ABB RAPID module: Target_R.mod

MODULE Target_R
    CONST robtarget TG_pick:=[[177.042141649,-272.000801516,190.000004036],[0.000000058,0.923879576,0.000000285,0.382683327],[0,-2,-1,4],[-107.239308648,9E+09,9E+09,9E+09,9E+09,9E+09]];
    CONST robtarget pick_up:=[[100.000104042,-278.500207981,150.000028222],[-0.000000126,-0.707106773,0.707106789,0.000000032],[0,-2,-1,4],[-101.964426672,9E+09,9E+09,9E+09,9E+09,9E+09]];
    CONST robtarget pick:=[[100,-278.5,50.43],[0,-0.707106781,0.707106781,0],[0,-2,-1,4],[-101.964426261,9E+09,9E+09,9E+09,9E+09,9E+09]];
    CONST robtarget check_BFR:=[[337.65,-25.09,414.16],[0.47949,-0.522281,0.486899,0.510138],[1,0,-1,4],[-166.865,9E+09,9E+09,9E+09,9E+09,9E+09]];
    CONST robtarget check_R:=[[352.06,-3.78,414.93],[0.468537,-0.49966,-0.504407,0.525725],[1,0,-2,4],[171.664,9E+09,9E+09,9E+09,9E+09,9E+09]];
    CONST robtarget TG_waitpoint:=[[260.000500472,-88.346067188,381.139966328],[0.499999312,-0.500000007,0.500000478,0.500000203],[0,0,-2,4],[-157.417353478,9E+09,9E+09,9E+09,9E+09,9E+09]];
    CONST robtarget waitpoint:=[[320.000617334,-110.201098524,199.999425349],[0.499999098,-0.500000027,0.500000616,0.50000026],[1,0,-1,4],[-162.867770325,9E+09,9E+09,9E+09,9E+09,9E+09]];
    CONST robtarget center:=[[320.000394297,-24.06071977,199.999617271],[0.499999361,-0.499999966,0.500000448,0.500000224],[1,0,-2,4],[-162.867771789,9E+09,9E+09,9E+09,9E+09,9E+09]];
    CONST robtarget home:=[[89.387954365,-156.622115869,147.913470331],[0.066010721,-0.842420916,-0.111214905,-0.523068666],[0,0,0,4],[-101.964426493,9E+09,9E+09,9E+09,9E+09,9E+09]];
    CONST robtarget TG_case_1:=[[320,-35.2,200],[0.5,-0.5,0.5,0.5],[1,0,-1,4],[-162.867772063,9E+09,9E+09,9E+09,9E+09,9E+09]];
    CONST robtarget TG_case_1_2:=[[285,-0.2,200],[0.707106781,0,0.707106781,0],[1,1,1,4],[-162.867775031,9E+09,9E+09,9E+09,9E+09,9E+09]];
    CONST robtarget TG_case_1_3:=[[250.000130819,-0.200197514,199.999945575],[0.707106719,-0.000000126,0.707106844,-0.000000064],[1,1,1,4],[-162.867770883,9E+09,9E+09,9E+09,9E+09,9E+09]];
    CONST robtarget TG_case_1_4:=[[250.000195865,-100.200387425,199.999831039],[0.707106608,-0.000000212,0.707106955,-0.000000105],[1,1,1,4],[-162.867770415,9E+09,9E+09,9E+09,9E+09,9E+09]];
    CONST robtarget pick_1_point:=[[320,-35.2,200],[0.707106781,-0.707106781,0,0],[1,0,-1,4],[-162.867772063,9E+09,9E+09,9E+09,9E+09,9E+09]];
    CONST robtarget TG_case_2_1:=[[320,-0.2,235],[0,1,0,0],[1,-1,-1,4],[-162.867775031,9E+09,9E+09,9E+09,9E+09,9E+09]];
    CONST robtarget TG_case_2_2:=[[320.00011125,-0.200157209,306.536956391],[0.000000065,1,0.000000052,-0.00000012],[1,-1,-1,4],[166.919278414,9E+09,9E+09,9E+09,9E+09,9E+09]];
    CONST robtarget TG_case_2_3:=[[320.000334899,-113.398256372,306.805846715],[-0.00000017,1,-0.000000477,0.000000268],[0,-1,-1,4],[166.919279952,9E+09,9E+09,9E+09,9E+09,9E+09]];
    CONST robtarget TG_case_6_1:=[[320.000434738,-150.200475591,260.570278198],[0.500000225,-0.500000005,0.49999967,0.5000001],[0,0,-2,4],[166.919277332,9E+09,9E+09,9E+09,9E+09,9E+09]];
    CONST robtarget TG_case_6_2:=[[320.000246228,-100.200299846,289.999834467],[-0.000000217,0.707106833,-0.707106729,-0.000000032],[0,-1,0,4],[166.919278031,9E+09,9E+09,9E+09,9E+09,9E+09]];
    CONST robtarget TG_case_6_3:=[[320.000112064,-0.200157006,289.999933843],[-0.000000136,0.707106819,-0.707106743,-0.00000002],[1,-1,0,4],[166.919275511,9E+09,9E+09,9E+09,9E+09,9E+09]];
    CONST robtarget TG_case_6:=[[320,-0.2,235],[0,-0.707106781,0.707106781,0],[1,-1,0,4],[-162.86777077,9E+09,9E+09,9E+09,9E+09,9E+09]];
    CONST robtarget TG_case_7_1:=[[320.000117939,-64.734463214,263.51272145],[0.000000148,0.707106808,-0.707106754,0.000000038],[1,-1,0,4],[-162.867775643,9E+09,9E+09,9E+09,9E+09,9E+09]];
    CONST robtarget TG_case_7:=[[320,-35.2,200],[0.5,-0.5,0.5,0.5],[1,0,-1,4],[-162.867774398,9E+09,9E+09,9E+09,9E+09,9E+09]];
    CONST robtarget TG_case_8:=[[355,-0.2,200],[0,-0.707106781,0,0.707106781],[1,-1,-1,4],[-162.867775031,9E+09,9E+09,9E+09,9E+09,9E+09]];
    CONST robtarget TG_case_8_1:=[[380.000103654,-0.200179059,199.999934552],[0.000000177,-0.707106678,-0.000000007,0.707106884],[1,-1,-1,4],[-162.86777415,9E+09,9E+09,9E+09,9E+09,9E+09]];
    CONST robtarget TG_case_8_2:=[[380.000209302,-100.200370788,199.999827465],[0.000000278,-0.707106534,0.000000011,0.707107029],[1,-1,-1,4],[-162.86777085,9E+09,9E+09,9E+09,9E+09,9E+09]];
    CONST robtarget TG_case_10:=[[320,-35.2,200],[0.707106781,-0.707106781,0,0],[1,0,2,4],[-162.867772063,9E+09,9E+09,9E+09,9E+09,9E+09]];
    CONST robtarget TG_case_10_1:=[[320.000696268,-90.201288322,199.99935497],[0.707106242,-0.707107321,0.000000473,0.000000897],[1,0,-1,4],[-162.867772063,9E+09,9E+09,9E+09,9E+09,9E+09]];
    CONST robtarget TG_case_13:=[[320.000100011,-0.200162708,234.999923315],[0.000000141,0.707106827,-0.707106735,-0.000000017],[1,-1,-1,4],[-162.867771316,9E+09,9E+09,9E+09,9E+09,9E+09]];
    CONST robtarget TG_case_13_1:=[[320.000219717,-0.200352952,289.999812905],[-0.000000351,0.707106881,-0.707106682,-0.000000022],[1,-1,0,4],[-162.867776998,9E+09,9E+09,9E+09,9E+09,9E+09]];
    CONST robtarget TG_case_13_2:=[[320.000309773,-100.200513401,289.999730794],[-0.000000495,0.707106929,-0.707106634,-0.000000033],[1,-1,0,4],[-162.86776981,9E+09,9E+09,9E+09,9E+09,9E+09]];
    CONST robtarget TG_case_15:=[[320.000221582,-0.200355951,234.999807219],[-0.000000301,-0.000000108,1,-0.000000207],[1,-1,1,4],[-162.867773678,9E+09,9E+09,9E+09,9E+09,9E+09]];
    CONST robtarget TG_case_15_1:=[[320.000304424,-0.200534501,289.99971144],[-0.000000436,-0.000000187,1,-0.000000319],[1,-1,1,4],[-162.86777685,9E+09,9E+09,9E+09,9E+09,9E+09]];
    CONST robtarget TG_case_15_2:=[[320.000420863,-100.200689662,289.999611172],[-0.000000567,-0.000000222,1,-0.000000412],[1,-1,1,4],[-162.867772341,9E+09,9E+09,9E+09,9E+09,9E+09]];
    CONST robtarget TG_case_16:=[[320.000100011,-0.200162708,234.999923315],[-0.000000112,-0.000000065,1,-0.000000088],[1,-1,1,4],[-162.867771316,9E+09,9E+09,9E+09,9E+09,9E+09]];
    CONST robtarget TG_case_16_1:=[[320.000219722,-0.200352952,289.999812905],[-0.000000263,-0.000000123,1,-0.000000232],[1,-1,1,4],[-162.867776998,9E+09,9E+09,9E+09,9E+09,9E+09]];
    CONST robtarget TG_case_16_2:=[[320.000316796,-100.20049956,289.999731895],[-0.000000438,-0.000000218,1,-0.000000304],[1,-1,1,4],[-162.867771749,9E+09,9E+09,9E+09,9E+09,9E+09]];
    CONST robtarget TG_case_17:=[[320.000100392,-70.200201954,199.999919618],[-0.000000103,0.000000037,0.707106889,0.707106674],[1,0,-1,4],[-162.867775031,9E+09,9E+09,9E+09,9E+09,9E+09]];
    CONST robtarget TG_case_24:=[[320.000088608,-135.200191217,199.999924774],[0.707106737,-0.707106825,0.000000199,0.000000049],[1,0,-1,4],[-162.867773249,9E+09,9E+09,9E+09,9E+09,9E+09]];
    CONST robtarget TG_case_2_4:=[[320.000193843,-113.398128068,306.805910112],[0.499999711,-0.499999999,0.500000151,0.500000139],[0,0,-2,4],[166.919276889,9E+09,9E+09,9E+09,9E+09,9E+09]];
    CONST robtarget rotate_B:=[[320.000078235,-0.200188226,223.859927266],[-0.000000157,-0.000000071,1,-0.000000117],[1,-1,1,4],[-162.867775813,9E+09,9E+09,9E+09,9E+09,9E+09]];
    CONST robtarget rotate_DUL:=[[320.000598398,-35.201112091,199.99943266],[0.499999079,-0.500000021,0.500000622,0.500000278],[1,0,-1,4],[-162.867770313,9E+09,9E+09,9E+09,9E+09,9E+09]];
    CONST robtarget TG_rotate_x2:=[[320.000670091,-104.963963276,199.999329246],[0.500000386,-0.500000721,-0.499999978,-0.499998916],[1,0,1,4],[-162.867773751,9E+09,9E+09,9E+09,9E+09,9E+09]];
    CONST robtarget rotate_F:=[[320,-0.2,223.86],[0,1,0,0],[1,-1,-1,4],[-162.867773629,9E+09,9E+09,9E+09,9E+09,9E+09]];
    CONST robtarget TG_check_BFR:=[[337.66,-153.73,414.06],[0.479377,-0.522264,0.486975,0.510191],[0,0,-1,4],[-166.857,9E+09,9E+09,9E+09,9E+09,9E+09]];
    CONST robtarget TG_rotate_CCW:=[[320.000820874,-100.201478448,199.9992449],[0.707106205,-0.707107357,0.000000517,0.000001213],[1,0,-1,4],[-162.867776692,9E+09,9E+09,9E+09,9E+09,9E+09]];
    CONST robtarget TG_rotate_CW:=[[320.000670091,-100.201293532,199.999329246],[-0.000001039,0.000000525,0.707107275,0.707106287],[1,0,-1,4],[-162.867773751,9E+09,9E+09,9E+09,9E+09,9E+09]];
ENDMODULE
